FUNCTION_BLOCK TcoStateTest EXTENDS TcoState
VAR
    _myIdentity : ULINT;
    _myContextIdentity : ULINT;
    _myContextStartCount : ULINT;
    _myContextEndCount : ULINT;
    _myParentIdentity : ULINT;
    _myState : INT;
    _tcoTaskTest_A : TcoTaskTest(THIS^);
    _tcoTaskTest_B : TcoTaskTest(THIS^);
    _tcoStateTest_A : TcoStateAutoRestoreTest(THIS^, eRestoreMode.None);
    _tcoStateTest_B : TcoStateAutoRestoreTest(THIS^, eRestoreMode.None);
    _onStateChangeCounter : INT;
    _autoRestoreToMyChildsEnabled : BOOL;
    _autoRestoreByMyParentEnabled : BOOL;
END_VAR

{attribute 'TcRpcEnable'}
METHOD INTERNAL CallTaskInstancies
_tcoTaskTest_A();
_tcoTaskTest_B();
END_METHOD

{attribute 'TcRpcEnable'}
METHOD INTERNAL CleanUp
THIS^.ChangeState(0);
_myState := State;
_onStateChangeCounter := 0;
_autoRestoreToMyChildsEnabled := FALSE;
_autoRestoreByMyParentEnabled := FALSE;
END_METHOD

{attribute 'TcRpcEnable'}
METHOD INTERNAL GetMessage : STRING
GetMessage := SUPER^._messenger._mime.Text;
END_METHOD

METHOD PROTECTED OnStateChange
VAR_INPUT
    PreviousState : INT;
    NewState : INT;
END_VAR
VAR
    message : STRING;
END_VAR
_onStateChangeCounter := _onStateChangeCounter + 1;
message := CONCAT('My state has been change from ', INT_TO_STRING(PreviousState));
message := CONCAT(message, ' to the new state ');
message := CONCAT(message, INT_TO_STRING(NewState));
message := CONCAT(message, '.');
THIS^.Messenger.Post(message, eMessageCategory.Debug);
SUPER^.OnStateChange(PreviousState, NewState);
END_METHOD

{attribute 'TcRpcEnable'}
METHOD INTERNAL PostMessage
VAR_INPUT
    Message : STRING;
END_VAR
THIS^.Messenger.Post(Message, eMessageCategory.Debug);
END_METHOD

{attribute 'TcRpcEnable'}
METHOD INTERNAL ReadOutAutoRestoreProperties
_autoRestoreToMyChildsEnabled := THIS^.IsAutoRestoreEnabled;
_autoRestoreByMyParentEnabled := THIS^.AutoRestorable;
END_METHOD

{attribute 'TcRpcEnable'}
METHOD INTERNAL ReadOutIdentities
_myIdentity := THIS^.Identity;
_myContextIdentity := THIS^.Context.Identity;
_myParentIdentity := THIS^.Parent.Identity;
_myContextStartCount := THIS^.Context.StartCycleCount;
_myContextEndCount := THIS^.Context.EndCycleCount;
END_METHOD

{attribute 'TcRpcEnable'}
METHOD INTERNAL ReadOutState
_myState := THIS^.State;
THIS^._tcoTaskTest_A.ReadOutState();
THIS^._tcoTaskTest_B.ReadOutState();
END_METHOD

{attribute 'TcRpcEnable'}
METHOD INTERNAL TriggerChangeState
VAR_INPUT
    NewState : INT;
END_VAR
THIS^.ChangeState(NewState);
END_METHOD

{attribute 'TcRpcEnable'}
METHOD INTERNAL TriggerChangeStateWithObjectRestore
VAR_INPUT
    NewState : INT;
END_VAR
THIS^.ChangeState(NewState).RestoreObject(THIS^._tcoTaskTest_A).RestoreObject(THIS^._tcoTaskTest_B);
END_METHOD

{attribute 'TcRpcEnable'}
METHOD INTERNAL TriggerRestore
THIS^.Restore();
END_METHOD

{attribute 'TcRpcEnable'}
METHOD INTERNAL TriggerTaskInvoke
THIS^._tcoTaskTest_A.Invoke();
THIS^._tcoTaskTest_B.Invoke();
END_METHOD

END_FUNCTION_BLOCK

(* stored: Version 1.1.0.1
   POU TcoStateTest: Id {efe977d1-c2f8-4084-8704-172d8704be2b}, SpecialFunc None
   Method CallTaskInstancies: Id {d3874270-1310-467f-9c2f-efa3788ae22b}
   Method CleanUp: Id {97d25468-22c5-42c9-8a2c-be94cbca7c7c}
   Method GetMessage: Id {7b51bd8a-afe2-4dba-b6f3-e076e50ff483}
   Method OnStateChange: Id {2efff8ba-6cfc-49c5-95bb-23754d8da191}
   Method PostMessage: Id {1cf19fab-faf4-4a89-aa3f-4a22ca64a534}
   Method ReadOutAutoRestoreProperties: Id {bc7f7afd-e36e-4b01-b682-4363a94409ab}
   Method ReadOutIdentities: Id {b63ec51a-adb3-49d9-99bc-5688aeb0dc91}
   Method ReadOutState: Id {5e78c467-c718-4bb6-9c71-a1bf248462a9}
   Method TriggerChangeState: Id {700ce7cc-dcaf-42d5-92d9-f568d5058a79}
   Method TriggerChangeStateWithObjectRestore: Id {20715526-f167-4822-9121-e7dd33bd0a9c}
   Method TriggerRestore: Id {e7cb051e-64b7-4a16-8b2b-2a6659a2020b}
   Method TriggerTaskInvoke: Id {b4293d91-dd5e-4ff8-a9d2-e2601a3de3ce} *)
